Universal Robots PolyScope program: motor_plate_full.urp

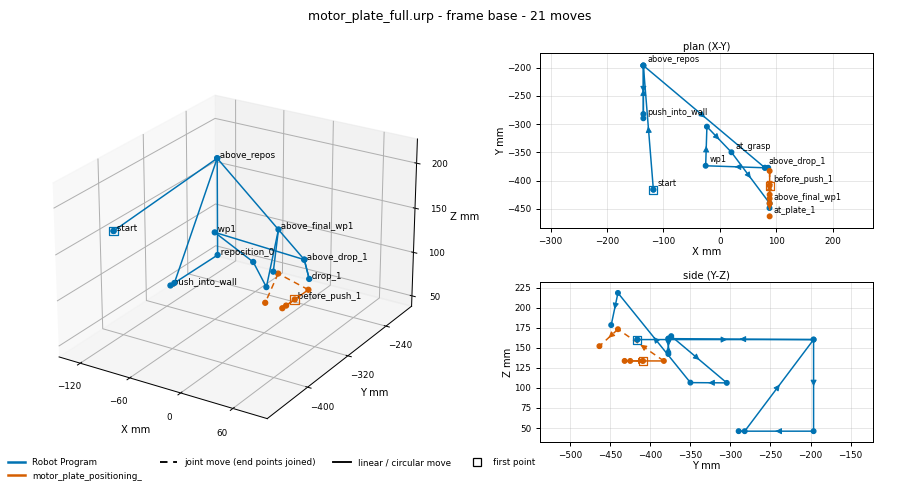
[picture p0: tool path of motor_plate_full.urp in frame base, 21 of 22 moves have a stored position in this frame; points joined in program order, loops and branches not executed]
Program motor_plate_full (installation=default directory=/programs/wrs2020 createdIn=5.6.0.90886 lastSavedIn=5.9.1.1031110 robotSerialNumber=20205500180)
Calibrated DH parameters: a=[0, -0.425, -0.3922, 0, 0, 0]; d=[0.1625, 0, 0, 0.1333, 0.0997, 0.0996]; alpha=[1.570796, 0, 0, 1.570796, -1.570796, 0]; deltaTheta=[0, 0, 0, 0, 0, 0]
Robot Program (runOnlyOnce=true)
  MoveJ speed 60 deg/s, acceleration 80 deg/s^2 (useActiveTCP=true) feature=Base
    currentpose := get_actual_tcp_pose()get_actual_joint_positions()
    Waypoint Waypoint (Variable): variable=currentpose
  SuppressedNode
    Folder Hardcoded pick
      MoveL speed 250 mm/s, acceleration 1200 mm/s^2 (useActiveTCP=true) feature=Base
        URCap Gripper (Robotiq_Grippers, Robotiq Inc.) dataModel(position=62.745098039215684, force=100.0, speed=100.0, positionInDouble=62.745098039215684, forceInDouble=100.0, speedInDouble=100.0, slaveIds=[9], blocking=true)
        Waypoint above_ex_pick: TCP in base x=-138.226 y=-538.226 z=142.964 mm, rx=-2.2047 ry=-2.2053 rz=0.0295 rad; joints [62.657, -81.157, 99.146, -108.621, -91.589, 62.632] deg; TCP offset x=0 y=0 z=220 mm, rx=0 ry=0 rz=0 rad
        Waypoint pick_plate: TCP in base x=-138.225 y=-538.241 z=68.355 mm, rx=-2.2047 ry=-2.2054 rz=0.0296 rad; joints [62.657, -77.051, 106.025, -119.611, -91.588, 62.632] deg
        URCap Gripper (Robotiq_Grippers, Robotiq Inc.) dataModel(position=100.0, force=0.0, speed=0.0, positionInDouble=100.0, forceInDouble=0.0, speedInDouble=0.0, slaveIds=[9], blocking=true)
  Folder Rearrange
    MoveJ speed 60 deg/s, acceleration 80 deg/s^2 (useActiveTCP=true) feature=Base
      Waypoint start: motionParameters(blendRadius=0.03); TCP in base x=-117.864 y=-415.957 z=160.266 mm, rx=2.1923 ry=2.2501 rz=0.0089 rad; joints [56.173, -98.859, 113.935, -104.756, -89.939, 54.684] deg
    MoveL speed 800 mm/s, acceleration 1200 mm/s^2 (useActiveTCP=false) tcp=gripper_140_tip; feature=Base
      Waypoint start: motionParameters(blendRadius=0.03); TCP in base x=-117.864 y=-415.957 z=160.266 mm, rx=2.1923 ry=2.2501 rz=0.0089 rad; joints [56.173, -98.859, 113.935, -104.756, -89.939, 54.684] deg
      Waypoint above_repos: motionParameters(blendRadius=0.05); TCP in base x=-135.607 y=-196.202 z=160.258 mm, rx=0.0308 ry=3.1376 rz=-0.0066 rad; joints [20.876, -133.857, 132.235, -88.26, -89.695, -68] deg; TCP offset x=0 y=0 z=220 mm, rx=0 ry=0 rz=0 rad
      Waypoint reposition_0: TCP in base x=-135.6 y=-196.2 z=46.036 mm, rx=0.0308 ry=3.1376 rz=-0.0066 rad; joints [20.876, -130.464, 148.282, -107.699, -89.695, -68] deg; TCP offset x=0 y=0 z=220 mm, rx=0 ry=0 rz=0 rad
      SuppressedNode
        URCap Gripper (Robotiq_Grippers, Robotiq Inc.) dataModel(position=72.54901960784314, force=0.0, speed=0.0, positionInDouble=72.54901960784314, forceInDouble=0.0, speedInDouble=0.0, slaveIds=[9], blocking=true)
      URCap Gripper (Robotiq_Grippers, Robotiq Inc.) dataModel(position=83.92156862745098, force=0.0, speed=0.0, positionInDouble=83.92156862745098, forceInDouble=0.0, speedInDouble=0.0, slaveIds=[9], blocking=true)
      Waypoint push_into_wall: TCP in base x=-135.617 y=-289.652 z=46.047 mm, rx=0.0296 ry=3.1376 rz=-0.0066 rad; joints [39.919, -110.73, 140.431, -119.691, -89.673, -49] deg; TCP offset x=0 y=0 z=220 mm, rx=0 ry=0 rz=0 rad
      URCap Gripper (Robotiq_Grippers, Robotiq Inc.) dataModel(position=72.54901960784314, force=0.0, speed=0.0, positionInDouble=72.54901960784314, forceInDouble=0.0, speedInDouble=0.0, slaveIds=[9], blocking=true)
      Waypoint regrasp1: TCP in base x=-135.585 y=-282.102 z=46.011 mm, rx=0.048 ry=3.1373 rz=-0.0065 rad; joints [38.754, -112.122, 141.194, -119.051, -89.674, -49.491] deg; TCP offset x=0 y=0 z=220 mm, rx=0 ry=0 rz=0 rad
      URCap Gripper (Robotiq_Grippers, Robotiq Inc.) dataModel(position=100.0, force=0.0, speed=0.0, positionInDouble=100.0, forceInDouble=0.0, speedInDouble=0.0, slaveIds=[9], blocking=true)
      Waypoint above_repos: TCP in base x=-135.607 y=-196.202 z=160.258 mm, rx=0.0308 ry=3.1376 rz=-0.0066 rad; joints [20.876, -133.857, 132.235, -88.26, -89.695, -68] deg; TCP offset x=0 y=0 z=220 mm, rx=0 ry=0 rz=0 rad
      URCap Gripper (Robotiq_Grippers, Robotiq Inc.) dataModel(position=100.0, force=0.0, speed=0.0, positionInDouble=100.0, forceInDouble=0.0, speedInDouble=0.0, slaveIds=[9], blocking=true)
  MoveL speed 800 mm/s, acceleration 1200 mm/s^2 (useActiveTCP=false) tcp=gripper_140_tip; feature=Base
    Waypoint above_drop_1: TCP in base x=79.695 y=-377.265 z=161.422 mm, rx=0.0416 ry=-3.1373 rz=-0.0063 rad; joints [81.935, -106.141, 119.316, -102.983, -90.263, -9.585] deg; TCP offset x=0 y=0 z=220 mm, rx=0 ry=0 rz=0 rad
    Waypoint drop_1: TCP in base x=85.464 y=-377.251 z=142.278 mm, rx=0.0417 ry=-3.1373 rz=-0.0063 rad; joints [82.835, -105.178, 121.536, -106.16, -90.26, -8.686] deg
    URCap Gripper (Robotiq_Grippers, Robotiq Inc.) dataModel(position=70.19607843137254, force=100.0, speed=100.0, positionInDouble=70.19607843137254, forceInDouble=100.0, speedInDouble=100.0, slaveIds=[9], blocking=true)
    Waypoint above_drop_1: TCP in base x=79.695 y=-377.265 z=161.422 mm, rx=0.0416 ry=-3.1373 rz=-0.0063 rad; joints [81.935, -106.141, 119.316, -102.983, -90.263, -9.585] deg
    Waypoint wp1: motionParameters(blendRadius=0.05); TCP in base x=-25.271 y=-373.698 z=164.531 mm, rx=0.4375 ry=2.7113 rz=-0.1186 rad; joints [44.743, -110.618, 123.094, -92.727, -69.038, -28.731] deg
    Waypoint before_grasp: motionParameters(blendRadius=0.02); TCP in base x=-23.072 y=-304.432 z=106.273 mm, rx=0.6188 ry=1.4761 rz=-0.6273 rad; joints [-14.061, -76.831, 148.353, -71.179, -58.369, -90.386] deg
    Waypoint at_grasp: TCP in base x=20.395 y=-349.807 z=106.586 mm, rx=0.6189 ry=1.4761 rz=-0.6273 rad; joints [-3.518, -79.015, 152.009, -72.602, -47.821, -90.469] deg
    URCap Gripper (Robotiq_Grippers, Robotiq Inc.) dataModel(position=100.0, force=100.0, speed=100.0, positionInDouble=100.0, forceInDouble=100.0, speedInDouble=100.0, slaveIds=[9], blocking=true)
    MoveDirectionNode (selectedDirection=ZPlus)
      Until DISTANCE (allowActions=false deceleration=3 distanceNodeType=BLEND) Distance=0.3; motionParameters(blendRadius=0.08)
    Waypoint above_final_wp1: motionParameters(blendRadius=0.03); TCP in base x=88.006 y=-440.155 z=218.409 mm, rx=0.0038 ry=3.0942 rz=-0.5375 rad; joints [81.985, -112.578, 122.706, -119.656, -87.271, -7.405] deg; TCP offset x=0 y=0 z=220 mm, rx=0 ry=0 rz=0 rad
    Waypoint final_1: TCP in base x=87.742 y=-448.558 z=178.336 mm, rx=0.001 ry=-2.8294 rz=1.3319 rad; joints [77.531, -118.839, 154.57, -175.58, -81.14, -8.388] deg; TCP offset x=0 y=0 z=220 mm, rx=0 ry=0 rz=0 rad
    URCap Gripper (Robotiq_Grippers, Robotiq Inc.) dataModel(position=70.19607843137254, force=100.0, speed=100.0, positionInDouble=70.19607843137254, forceInDouble=100.0, speedInDouble=100.0, slaveIds=[9], blocking=true)
    URCap Gripper (Robotiq_Grippers, Robotiq Inc.) dataModel(position=100.0, force=0.0, speed=0.0, positionInDouble=100.0, forceInDouble=0.0, speedInDouble=0.0, slaveIds=[9], blocking=true)
    URCap Gripper (Robotiq_Grippers, Robotiq Inc.) dataModel(position=70.19607843137254, force=100.0, speed=100.0, positionInDouble=70.19607843137254, forceInDouble=100.0, speedInDouble=100.0, slaveIds=[9], blocking=true)
  Call motor_plate_positioning_1
SubProgram -> motor_plate_positioning_1
SubProgram motor_plate_positioning_1 (keepSynchronizedWithDisk=false) programFile=/programs/wrs2020/motor_plate_positioning.urp
  MoveL speed 250 mm/s, acceleration 1200 mm/s^2 (useActiveTCP=false) tcp=gripper_140_tip; feature=Base
    Waypoint before_push_1: TCP in base x=88.025 y=-408.839 z=133.608 mm, rx=0.004 ry=3.1409 rz=-0.0122 rad; joints [83.494, -100.382, 119.446, -109.501, -89.913, -6.359] deg
  URCap Gripper (Robotiq_Grippers, Robotiq Inc.) dataModel(position=100.0, force=0.0, speed=0.0, positionInDouble=100.0, forceInDouble=0.0, speedInDouble=0.0, slaveIds=[9], blocking=true)
  MoveL speed 250 mm/s, acceleration 1200 mm/s^2 (useActiveTCP=false) tcp=gripper_140_tip; feature=Base
    Waypoint push_almost_end: motionParameters(jointSpeed=1.047198 jointAcceleration=1.396263 cartesianSpeed=0.1 cartesianAcceleration=0.1 blendRadius=0.004); TCP in base x=88.002 y=-424.84 z=133.627 mm, rx=0.004 ry=3.141 rz=0.0085 rad; joints [83.81, -97.445, 116.826, -109.071, -90, -6.046] deg
    Waypoint push_end_1: motionParameters(jointSpeed=1.047198 jointAcceleration=1.396263 cartesianSpeed=0.05 cartesianAcceleration=0.008); TCP in base x=87.978 y=-431.827 z=133.657 mm, rx=0.0041 ry=3.1408 rz=-0.0293 rad; joints [83.796, -97.423, 117.18, -110.815, -89.851, -6.053] deg
    Waypoint before_push_2: motionParameters(jointSpeed=1.047198 jointAcceleration=1.396263 cartesianSpeed=0.8 cartesianAcceleration=0.8); TCP in base x=88.017 y=-382.896 z=133.609 mm, rx=0.004 ry=3.1409 rz=-0.0122 rad; joints [83.034, -104.382, 122.465, -108.52, -89.91, -6.818] deg
  URCap Gripper (Robotiq_Grippers, Robotiq Inc.) dataModel(position=70.19607843137254, force=100.0, speed=100.0, positionInDouble=70.19607843137254, forceInDouble=100.0, speedInDouble=100.0, slaveIds=[9], blocking=true)
  MoveJ speed 150 deg/s, acceleration 150 deg/s^2 (useActiveTCP=false) tcp=gripper_140_tip; feature=Base
    Waypoint above_plate_1: motionParameters(blendRadius=0.03); TCP in base x=88.01 y=-440.155 z=173.172 mm, rx=0.0038 ry=3.0942 rz=-0.5374 rad; joints [81.985, -110.774, 128.458, -127.209, -87.271, -7.405] deg
    Waypoint at_plate_1: TCP in base x=88.005 y=-463.265 z=152.055 mm, rx=0.0034 ry=2.946 rz=-1.087 rad; joints [79.411, -112.569, 147.397, -164.842, -83.11, -7.945] deg
  URCap Gripper (Robotiq_Grippers, Robotiq Inc.) dataModel(position=100.0, force=0.0, speed=0.0, positionInDouble=100.0, forceInDouble=0.0, speedInDouble=0.0, slaveIds=[9], blocking=true)
  URCap Gripper (Robotiq_Grippers, Robotiq Inc.) dataModel(position=82.3529411764706, force=100.0, speed=0.0, positionInDouble=82.3529411764706, forceInDouble=100.0, speedInDouble=0.0, slaveIds=[9], blocking=true)
